FUNCTION_BLOCK TEST_CLT (* Test Java emitter code generation for all kinds of I/O connections *)
  (* Standard: 61499-2 *)
  (* Version 0.0, 2004-01-02, JHC, Rockwell Automation *)
  (* Compiler header: package fb.rt.test; import fb.rt.net.*; *)
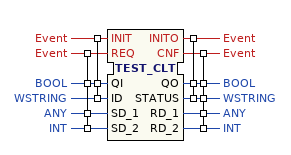
  EVENT_INPUT
    INIT WITH QI, ID; (* Initialize/Terminate *)
    REQ WITH QI, SD_1, SD_2; (* Send Request *)
  END_EVENT
  EVENT_OUTPUT
    INITO WITH QO, STATUS; (* Initialized/Terminated *)
    CNF WITH QO, STATUS, RD_1, RD_2; (* Data Received/Error *)
  END_EVENT
  VAR_INPUT
    QI : BOOL; (* Input event qualifier *)
    ID : WSTRING;
    SD_1 : ANY;
    SD_2 : INT;
  END_VAR
  VAR_OUTPUT
    QO : BOOL; (* Output event qualifier *)
    STATUS : WSTRING;
    RD_1 : ANY;
    RD_2 : INT;
  END_VAR
  FBS
    CLT : CLIENT_2;
  END_FBS
  EVENT_CONNECTIONS
    INIT TO CLT.INIT;
    REQ TO CLT.REQ;
    CLT.INITO TO INITO;
    CLT.CNF TO CNF;
  END_CONNECTIONS
  DATA_CONNECTIONS
    QI TO CLT.QI;
    ID TO CLT.ID;
    SD_1 TO CLT.SD_1;
    SD_2 TO CLT.SD_2;
    CLT.QO TO QO;
    CLT.STATUS TO STATUS;
    CLT.RD_1 TO RD_1;
    CLT.RD_2 TO RD_2;
  END_CONNECTIONS
END_FUNCTION_BLOCK
